// TwinCAT 3 PLC project PLC
// ProgramVersion: 3.1.4026.20
// CompilerDefines: VISU_USEPROPERTYINFO
// libraries:
//   SPT Base Types, * (Beckhoff Automation LLC)
//   SPT Components, * (Beckhoff Automation LLC)
//   SPT Diagnostic, * (Beckhoff Automation LLC)
//   SPT EtherCat, * (Beckhoff Automation LLC)
//   SPT Event Logger, * (Beckhoff Automation LLC)
//   SPT Motion Control, * (Beckhoff Automation LLC)
//   SPT Utilities, * (Beckhoff Automation LLC)
//   Tc2_MC2, * (Beckhoff Automation GmbH)
//   Tc2_MC2_Camming, * (Beckhoff Automation GmbH)
//   Tc2_Standard, * (Beckhoff Automation GmbH)
//   Tc2_System, * (Beckhoff Automation GmbH)
//   Tc2_Utilities, * (Beckhoff Automation GmbH)
//   Tc3_EventLogger, * (Beckhoff Automation GmbH)
//   Tc3_MC2_AdvancedHoming, * (Beckhoff Automation GmbH)
//   Tc3_McCollisionAvoidance, * (Beckhoff Automation GmbH)
//   Tc3_McCoordinatedMotion, * (Beckhoff Automation GmbH)
//   Tc3_PackML_V3, * (Beckhoff Automation GmbH)
// project tree:
//   / GlobalTextList.TcGTLO (not stored), PlcTask.TcTTO (not stored), VisualizationManager.TcVMO (not stored)
//   GVLs/ GVL.TcGVL (not stored)
//   POUs/ Machine.TcPOU, MAIN.TcPOU (not stored)
//   POUs/RackAndPinion/ FB_RackAndPinion.TcPOU
//   VISUs/ Visualization.TcVIS (not stored)
// real-time tasks:
//   TASK PlcTask: cycle T#1ms, priority 20, ADS port 350
//   TASK Job Task: cycle default, priority 32
// motion (NC):
//   TASK NC-Task 1 SAF: cycle T#2ms, priority 4, ADS port 501
//   TASK NC-Task 1 SVB: cycle T#10ms, priority 8, ADS port 511
//   AXIS RnP_Left (id 1)
//     Dynamic: Acceleration=11599.5, Deceleration=11599.5, Jerk=34798.6
//     Velo: RefSearch=10, RefSync=10, SlowManual=1, FastManual=10, Fast=7733.014, Maximum=7733.01
//     OtherSettings: AllowMotionCmdToSlave=true
//     encoder EncType=19
//       EncPara: ScaleFactorNumerator=169.6464, ScaleFactorDenominator=1048576, MaxCount=#xffffffff
//         Inc: RefSearchInverse=true, RefSyncInverse=false, RefPosition=20, RefMode=1
//     drive DrvType=16
//       DrvPara: MaxCount=#xffffffff, DriveControlDWord=#x00020100
//         Analog: VeloReferenz=8506.3154, VeloScale=71.5255737304688, TorqueSetpointScale=10, ScaleFactorActTorque=0.1
//         TimeComp: TaskDelayCycles=1
//     controller CtrType=1
//       CtrPara: PriorControlFactor=1
//         PosDiffControl: Range=15
//         Observer: BandWidth=20
//   AXIS RnP_Right (id 2)
//     Dynamic: Acceleration=11599.521, Deceleration=11599.521, Jerk=34798.563
//     Velo: RefSearch=10, RefSync=10, SlowManual=1, FastManual=10, Fast=7733.014, Maximum=7733.014
//     OtherSettings: AllowMotionCmdToSlave=true
//     encoder EncType=19
//       EncPara: ScaleFactorNumerator=169.6464, ScaleFactorDenominator=1048576, MaxCount=#xffffffff
//         Inc: RefPosition=490, RefMode=6
//     drive DrvType=16
//       DrvPara: MaxCount=#xffffffff, DriveControlDWord=#x00020100
//         Analog: VeloReferenz=8506.3154, VeloScale=71.5255737304688, TorqueSetpointScale=10, ScaleFactorActTorque=0.1
//         TimeComp: TaskDelayCycles=1
//     controller CtrType=1
//       CtrPara: PriorControlFactor=1
//         PosDiffControl: Range=15
//         Observer: BandWidth=20
//   AXIS Ballscrew (id 3)
//     OtherSettings: AllowMotionCmdToSlave=true
//     encoder EncType=19
//       EncPara: MaxCount=#xffffffff
//     drive DrvType=16
//       DrvPara: MaxCount=#xffffffff, DriveControlDWord=#x00000100
//         Analog: TorqueSetpointScale=10, ScaleFactorActTorque=0.1
//         TimeComp: TaskDelayCycles=1
//     controller CtrType=1
//       CtrPara: PriorControlFactor=1
//         Observer: BandWidth=20
// I/O:
//   DEVICE Device 1 (EtherCAT), AmsNetId 169.254.243.188.2.1
//     Term 1 (EK1101) [EK1101 EtherCAT Coupler (2A E-Bus, ID switch)]
//       Term 2 (EL1904) [EL1904, 4 Ch. Safety Input 24V, TwinSAFE]
//         modules: Module 1 (FSOES)
//       Term 3 (EK1110) [EK1110 EtherCAT extension]
//     Term 4 (AX8620-0000-0105) [AX8620-0000-0105]
//       Drive 5 (AX8206-0210-0107) [AX8206-0210-0107 (2Ch. 6A servo axis, safe-motion, multi-FB)]
//         modules: Device, Device, Device, Device, Device, Device, Device, Device, Device, Device, Device (Safety), Device, Device, Device, Device, Device, Device, Device, Device, Device, Device, Device, Device, Device, Device, Device, Device, Device, Device, Device, Device, Ch A, Ch A, Ch A, Ch A, Ch A, Ch A, Ch A, Ch A, Ch A, Ch A, Ch A, Ch A, Ch A, Ch A, Ch A, Ch A, Ch A, Ch A, Ch A, Ch A, Ch A, Ch A, Ch A, Ch A, Ch A, Ch A, Ch B, Ch B, Ch B, Ch B, Ch B, Ch B, Ch B, Ch B, Ch B, Ch B, Ch B, Ch B, Ch B, Ch B, Ch B, Ch B, Ch B, Ch B, Ch B, Ch B, Ch B, Ch B, Ch B, Ch B, Ch B
//         startup 12992:1 := 414D383132312D78467830 // Ch A SynchronousMotor parameters / Configured motor type
//         startup 24768:0 := FEFF // Ch A Interpolation sub mode select
//         startup 13000:5 := 0200 // Ch A SynchronousMotor thermal model / Reaction
//         startup 13000:6 := 0000C841 // Ch A SynchronousMotor thermal model / Partial fraction factor
//         startup 12992:12 := 00803B45 // Ch A SynchronousMotor parameters / Motor rated speed
//         startup 12992:13 := 0000003F // Ch A SynchronousMotor parameters / Motor rated torque
//         startup 24694:0 := F4010000 // Ch A Motor standstill torque
//         startup 24800:0 := D007 // Ch A Positive torque/force limit value
//         startup 24801:0 := D007 // Ch A Negative torque/force limit value
//         startup 12288:6 := 4158383230362D303231302D30303030 // Ch A AxisMain parameters / Configured drive type
//         startup 12867:1 := 00008040 // Ch A TorqueControl parameters / Configured channel rated current
//         startup 12867:2 := 00004041 // Ch A TorqueControl parameters / Configured channel peak current
//         startup 12867:7 := 77BE1F40 // Ch A TorqueControl parameters / Iuvw max sum
//         startup 24672:0 := 08 // Ch A Modes of operation
//         startup 13023:0 := 0000 // Ch A SynchronousMotor control mode
//         startup 12998:1 := CDCCCC3C // Ch A SynchronousMotor commutation monitoring parameters / Speed threshold
//         startup 12864:1 := CAAD2041 // Ch A TorqueControl parameters mappable / Torque control proportional gain q
//         startup 12864:2 := 8A0E7C39 // Ch A TorqueControl parameters mappable / Torque control integral action time q
//         startup 12608:1 := FBD1CD3B // Ch A VelocityControl parameters mappable / Velocity control proportional gain
//         startup 12608:2 := 6F12033C // Ch A VelocityControl parameters mappable / Velocity control integral action time
//         startup 12608:3 := 00980546 // Ch A VelocityControl parameters mappable / Bipolar velocity limit value
//         startup 12992:15 := 0100 // Ch A SynchronousMotor parameters / Motor temperature sensor connection
//         startup 12611:4 := 0400 // Ch A VelocityControl observer / Observer type
//         startup 24672:0 := 08 // Ch A Modes of operation
//         startup 12296:2 := 00 // Ch A AxisMain parameters encoder direction / Primary encoder direction
//       Drive 6 (AX8206-0200-0106) [AX8206-0200-0106 (2Ch. 6A servo axis, safe-motion)]
//         modules: Device, Device, Device, Device, Device, Device, Device, Device, Device, Device, Device (Safety), Device, Device, Device, Device, Device, Device, Device, Device, Device, Device, Device, Device, Device, Device, Device, Device, Device, Device, Device, Device, Ch A, Ch A, Ch A, Ch A, Ch A, Ch A, Ch A, Ch A, Ch A, Ch A, Ch A, Ch A, Ch A, Ch A, Ch A, Ch A, Ch A, Ch A, Ch A, Ch A, Ch A, Ch A, Ch A, Ch A, Ch A, Ch A, Ch A, Ch B, Ch B, Ch B, Ch B, Ch B, Ch B, Ch B, Ch B, Ch B, Ch B, Ch B, Ch B, Ch B, Ch B, Ch B, Ch B, Ch B, Ch B, Ch B, Ch B, Ch B, Ch B, Ch B, Ch B, Ch B, Ch B, Ch B
//         startup 12992:1 := 414D383032322D78447831 // Ch A Motor parameters / Configured motor type
//         startup 24768:0 := FEFF // Ch A Interpolation sub mode select
//         startup 13000:5 := 0200 // Ch A Motor thermal model / Reaction
//         startup 13000:6 := 0000C841 // Ch A Motor thermal model / Partial fraction factor
//         startup 12992:12 := 0000FA45 // Ch A Motor parameters / Motor rated speed
//         startup 12992:13 := E561313F // Ch A Motor parameters / Motor rated torque
//         startup 24694:0 := 20030000 // Ch A Motor standstill torque
//         startup 24800:0 := D007 // Ch A Positive torque/force limit value
//         startup 24801:0 := D007 // Ch A Negative torque/force limit value
//         startup 12288:6 := 4158383230362D303230302D30303030 // Ch A AxisMain parameters / Configured drive type
//         startup 12867:1 := 0000C03F // Ch A TorqueCtrl parameters / Configured channel rated current
//         startup 12867:2 := 00009040 // Ch A TorqueCtrl parameters / Configured channel peak current
//         startup 12867:7 := 77BE1F40 // Ch A TorqueCtrl parameters / Iuvw max sum
//         startup 24672:0 := 08 // Ch A Modes of operation
//         startup 13023:0 := 0000 // Ch A Motor control mode
//         startup 12998:2 := 5D481A3D // Ch A Motor commutation monitoring parameters / Voltage threshold
//         startup 12998:1 := D5B01E3C // Ch A Motor commutation monitoring parameters / Speed threshold
//         startup 12864:1 := 88E9D742 // Ch A TorqueCtrl parameters mappable / Torque control proportional gain q
//         startup 12864:2 := 8A0E7C39 // Ch A TorqueCtrl parameters mappable / Torque control integral action time q
//         startup 12608:1 := 7298793C // Ch A VeloCtrl parameters mappable / Velocity control proportional gain
//         startup 12608:2 := 6F12033C // Ch A VeloCtrl parameters mappable / Velocity control integral action time
//         startup 12608:3 := 00980546 // Ch A VeloCtrl parameters mappable / Bipolar velocity limit value
//         startup 12992:15 := 0100 // Ch A Motor parameters / Motor temperature sensor connection
//         startup 12611:4 := 0400 // Ch A VeloCtrl observer / Observer type
//         startup 24672:0 := 08 // Ch A Modes of operation
//         startup 12296:2 := 00 // Ch A AxisMain parameters encoder direction / Primary encoder direction
//         startup 14016:1 := 414D383032322D78447831 // Ch B Motor parameters / Configured motor type
//         startup 26816:0 := FEFF // Ch B Interpolation sub mode select
//         startup 14024:5 := 0200 // Ch B Motor thermal model / Reaction
//         startup 14024:6 := 0000C841 // Ch B Motor thermal model / Partial fraction factor
//         startup 14016:12 := 0000FA45 // Ch B Motor parameters / Motor rated speed
//         startup 14016:13 := E561313F // Ch B Motor parameters / Motor rated torque
//         startup 26742:0 := 20030000 // Ch B Motor standstill torque
//         startup 26848:0 := D007 // Ch B Positive torque/force limit value
//         startup 26849:0 := D007 // Ch B Negative torque/force limit value
//         startup 13312:6 := 4158383230362D303230302D30303030 // Ch B AxisMain parameters / Configured drive type
//         startup 13891:1 := 0000C03F // Ch B TorqueCtrl parameters / Configured channel rated current
//         startup 13891:2 := 00009040 // Ch B TorqueCtrl parameters / Configured channel peak current
//         startup 13891:7 := 77BE1F40 // Ch B TorqueCtrl parameters / Iuvw max sum
//         startup 26720:0 := 08 // Ch B Modes of operation
//         startup 14047:0 := 0000 // Ch B Motor control mode
//         startup 14022:2 := 5D481A3D // Ch B Motor commutation monitoring parameters / Voltage threshold
//         startup 14022:1 := D5B01E3C // Ch B Motor commutation monitoring parameters / Speed threshold
//         startup 13888:1 := 88E9D742 // Ch B TorqueCtrl parameters mappable / Torque control proportional gain q
//         startup 13888:2 := 8A0E7C39 // Ch B TorqueCtrl parameters mappable / Torque control integral action time q
//         startup 13632:1 := 7298793C // Ch B VeloCtrl parameters mappable / Velocity control proportional gain
//         startup 13632:2 := 6F12033C // Ch B VeloCtrl parameters mappable / Velocity control integral action time
//         startup 13632:3 := 00980546 // Ch B VeloCtrl parameters mappable / Bipolar velocity limit value
//         startup 14016:15 := 0100 // Ch B Motor parameters / Motor temperature sensor connection
//         startup 13635:4 := 0400 // Ch B VeloCtrl observer / Observer type
//         startup 26720:0 := 08 // Ch B Modes of operation
//         startup 13320:2 := 00 // Ch B AxisMain parameters encoder direction / Primary encoder direction
// variable links:
//   NC-Task 1 SAF/Axes/RnP_Left <-> Device 1 (EtherCAT)/Term 4 (AX8620-0000-0105)/Drive 6 (AX8206-0200-0106)
//     Drive/Inputs/In/nDataIn1 <-> Ch A/Ch A PositionControl Inputs/Ch A Following error actual value
//     Drive/Inputs/In/nDataIn3[0] <-> Ch A/Ch A TorqueControl Inputs/Ch A Torque/force actual value
//     Drive/Inputs/In/nDcOutputTime <-> InfoData/DcOutputShift
//     Drive/Inputs/In/nState1 <-> Ch A/Ch A AxisMain Inputs/Ch A Statusword
//     Drive/Inputs/In/nState2 <-> Ch A/Ch A AxisMain Inputs/Ch A Statusword @bit 8
//     Drive/Inputs/In/nState4 @bit 1 <-> WcState/InputToggle0
//     Drive/Inputs/In/nState4 <-> WcState/WcState0
//     Drive/Outputs/Out/nCtrl1 <-> Ch A/Ch A AxisMain Outputs/Ch A Controlword
//     Drive/Outputs/Out/nCtrl2 <-> Ch A/Ch A AxisMain Outputs/Ch A Controlword @bit 8
//     Drive/Outputs/Out/nDataOut1 <-> Ch A/Ch A Interpolator Outputs/Ch A Target position
//     Drive/Outputs/Out/nDataOut2 <-> Ch A/Ch A Interpolator Outputs/Ch A Target velocity
//     Enc/Inputs/In/nDataIn1 <-> Ch A/Ch A AxisMain Inputs/Ch A Position actual value
//     Enc/Inputs/In/nDcInputTime <-> InfoData/DcInputShift
//     Enc/Inputs/In/nState2 @bit 5 <-> Ch A/Ch A AxisMain Inputs/Position actual value invalid
//     Enc/Inputs/In/nState4 @bit 1 <-> WcState/InputToggle0
//     Enc/Inputs/In/nState4 <-> WcState/WcState0
//   NC-Task 1 SAF/Axes/RnP_Right <-> Device 1 (EtherCAT)/Term 4 (AX8620-0000-0105)/Drive 6 (AX8206-0200-0106)
//     Drive/Inputs/In/nDataIn1 <-> Ch B/Ch B PositionControl Inputs/Ch B Following error actual value
//     Drive/Inputs/In/nDataIn3[0] <-> Ch B/Ch B TorqueControl Inputs/Ch B Torque/force actual value
//     Drive/Inputs/In/nDcOutputTime <-> InfoData/DcOutputShift
//     Drive/Inputs/In/nState1 <-> Ch B/Ch B AxisMain Inputs/Ch B Statusword
//     Drive/Inputs/In/nState2 <-> Ch B/Ch B AxisMain Inputs/Ch B Statusword @bit 8
//     Drive/Inputs/In/nState4 @bit 1 <-> WcState/InputToggle0
//     Drive/Inputs/In/nState4 <-> WcState/WcState0
//     Drive/Outputs/Out/nCtrl1 <-> Ch B/Ch B AxisMain Outputs/Ch B Controlword
//     Drive/Outputs/Out/nCtrl2 <-> Ch B/Ch B AxisMain Outputs/Ch B Controlword @bit 8
//     Drive/Outputs/Out/nDataOut1 <-> Ch B/Ch B Interpolator Outputs/Ch B Target position
//     Drive/Outputs/Out/nDataOut2 <-> Ch B/Ch B Interpolator Outputs/Ch B Target velocity
//     Enc/Inputs/In/nDataIn1 <-> Ch B/Ch B AxisMain Inputs/Ch B Position actual value
//     Enc/Inputs/In/nDcInputTime <-> InfoData/DcInputShift
//     Enc/Inputs/In/nState2 @bit 5 <-> Ch B/Ch B AxisMain Inputs/Position actual value invalid
//     Enc/Inputs/In/nState4 @bit 1 <-> WcState/InputToggle0
//     Enc/Inputs/In/nState4 <-> WcState/WcState0
//   PLC/PLC Instance <-> Device 1 (EtherCAT)/Term 4 (AX8620-0000-0105)/Drive 5 (AX8206-0210-0107)
//     PlcTask Inputs/MAIN.SafetyEstop.InfoData/Diag <-> Device (Safety)/Function Block Info Data/TwinSafeGroup1.Network1.FBEstop1 Info Data/Diag
//     PlcTask Inputs/MAIN.SafetyEstop.InfoData/State <-> Device (Safety)/Function Block Info Data/TwinSafeGroup1.Network1.FBEstop1 Info Data/State
//     PlcTask Inputs/MAIN.SafetyGroup_Main.InfoData/Diag <-> Device (Safety)/Group Info Data/TwinSafeGroup1 Info Data/Diag
//     PlcTask Inputs/MAIN.SafetyGroup_Main.InfoData/State <-> Device (Safety)/Group Info Data/TwinSafeGroup1 Info Data/State
//     PlcTask Inputs/MAIN.SafetyOK <-> Device (Safety)/Standard Inputdata/Standard Out Var 7
//     PlcTask Outputs/MAIN.SafetyFBReset <-> Device (Safety)/Standard Outputdata/Standard In Var 6
//     PlcTask Outputs/MAIN.SafetyGroupAutoReset.Reset <-> Device (Safety)/Standard Outputdata/Standard In Var 1
//     PlcTask Outputs/MAIN.SafetyGroup_Main.Run <-> Device (Safety)/Standard Outputdata/Standard In Var 2
//   PLC/PLC Instance <-> NC-Task 1 SAF/Axes/RnP_Left
//     PlcTask Inputs/MAIN.Machine.RackAndPinion.LeftAxis.BasicAxis._Axis.NcToPlc <-> Outputs/ToPlc
//     PlcTask Outputs/MAIN.Machine.RackAndPinion.LeftAxis.BasicAxis._Axis.PlcToNc <-> Inputs/FromPlc
//   PLC/PLC Instance <-> NC-Task 1 SAF/Axes/RnP_Right
//     PlcTask Inputs/MAIN.Machine.RackAndPinion.RightAxis.BasicAxis._Axis.NcToPlc <-> Outputs/ToPlc
//     PlcTask Outputs/MAIN.Machine.RackAndPinion.RightAxis.BasicAxis._Axis.PlcToNc <-> Inputs/FromPlc
//   PLC/PLC Instance <-> NC-Task 1 SAF/Objects/Group1 (CA Group)
//     PlcTask Inputs/MAIN.Machine.RackAndPinion.CAGroup.NcToPlc <-> Group Outputs/ToPLC
//     PlcTask Outputs/MAIN.Machine.RackAndPinion.CAGroup.PlcToNc/CA <-> Group Inputs/FromPLC
//   (this object) <-> Device 1 (EtherCAT)/Term 4 (AX8620-0000-0105)/Drive 5 (AX8206-0210-0107)
//     Drive/Inputs/In/nDataIn1 <-> Ch A/Ch A PositionControl Inputs/Ch A Following error actual value
//     Drive/Inputs/In/nDataIn3[0] <-> Ch A/Ch A TorqueControl Inputs/Ch A Torque/force actual value
//     Drive/Inputs/In/nDcOutputTime <-> InfoData/DcOutputShift
//     Drive/Inputs/In/nState1 <-> Ch A/Ch A AxisMain Inputs/Ch A Statusword
//     Drive/Inputs/In/nState2 <-> Ch A/Ch A AxisMain Inputs/Ch A Statusword @bit 8
//     Drive/Inputs/In/nState4 @bit 1 <-> WcState/InputToggle0
//     Drive/Inputs/In/nState4 <-> WcState/WcState0
//     Drive/Outputs/Out/nCtrl1 <-> Ch A/Ch A AxisMain Outputs/Ch A Controlword
//     Drive/Outputs/Out/nCtrl2 <-> Ch A/Ch A AxisMain Outputs/Ch A Controlword @bit 8
//     Drive/Outputs/Out/nDataOut1 <-> Ch A/Ch A Interpolator Outputs/Ch A Target position
//     Drive/Outputs/Out/nDataOut2 <-> Ch A/Ch A Interpolator Outputs/Ch A Target velocity
//     Enc/Inputs/In/nDataIn1 <-> Ch A/Ch A AxisMain Inputs/Ch A Position actual value
//     Enc/Inputs/In/nDcInputTime <-> InfoData/DcInputShift
//     Enc/Inputs/In/nState2 @bit 5 <-> Ch A/Ch A AxisMain Inputs/Position actual value invalid
//     Enc/Inputs/In/nState4 @bit 1 <-> WcState/InputToggle0
//     Enc/Inputs/In/nState4 <-> WcState/WcState0
//   (this object) <-> Device 1 (EtherCAT)
//     Term 1 (EK1101)/Term 2 (EL1904)/Module 1 (FSOES)/RxPDO/FSOE <-> Term 4 (AX8620-0000-0105)/Drive 5 (AX8206-0210-0107)/Device (Safety)/FSoE Master Connection 1 Master Message/Message_3
//     Term 1 (EK1101)/Term 2 (EL1904)/Module 1 (FSOES)/TxPDO/FSOE <-> Term 4 (AX8620-0000-0105)/Drive 5 (AX8206-0210-0107)/Device (Safety)/FSoE Master Connection 1 Slave Message/Message_3
//     Term 4 (AX8620-0000-0105)/Drive 5 (AX8206-0210-0107)/Device (Safety)/FSoE Master Connection 1 Master Message/Message_3 <-> Term 1 (EK1101)/Term 2 (EL1904)/Module 1 (FSOES)/RxPDO/FSOE
//     Term 4 (AX8620-0000-0105)/Drive 5 (AX8206-0210-0107)/Device (Safety)/FSoE Master Connection 1 Slave Message/Message_3 <-> Term 1 (EK1101)/Term 2 (EL1904)/Module 1 (FSOES)/TxPDO/FSOE
//     Term 4 (AX8620-0000-0105)/Drive 5 (AX8206-0210-0107)/Device (Safety)/FSoE Master Connection 2 Master Message/Message_5 <-> Term 4 (AX8620-0000-0105)/Drive 6 (AX8206-0200-0106)/Device (Safety)/FSoE Slave Connection 1 Master Message/FSOE
//     Term 4 (AX8620-0000-0105)/Drive 5 (AX8206-0210-0107)/Device (Safety)/FSoE Master Connection 2 Slave Message/Message_5 <-> Term 4 (AX8620-0000-0105)/Drive 6 (AX8206-0200-0106)/Device (Safety)/FSoE Slave Connection 1 Slave Message/FSOE
//     Term 4 (AX8620-0000-0105)/Drive 5 (AX8206-0210-0107)/Device/DeviceMain Outputs/Power supply controlword <-> Term 4 (AX8620-0000-0105)/PSM Controlword for axis/Controlword for axis
//     Term 4 (AX8620-0000-0105)/Drive 6 (AX8206-0200-0106)/Device/DeviceMain Outputs/Power supply controlword <-> Term 4 (AX8620-0000-0105)/PSM Controlword for axis/Controlword for axis
//     Term 4 (AX8620-0000-0105)/Drive 6 (AX8206-0200-0106)/Device (Safety)/FSoE Slave Connection 1 Master Message/FSOE <-> Term 4 (AX8620-0000-0105)/Drive 5 (AX8206-0210-0107)/Device (Safety)/FSoE Master Connection 2 Master Message/Message_5
//     Term 4 (AX8620-0000-0105)/Drive 6 (AX8206-0200-0106)/Device (Safety)/FSoE Slave Connection 1 Slave Message/FSOE <-> Term 4 (AX8620-0000-0105)/Drive 5 (AX8206-0210-0107)/Device (Safety)/FSoE Master Connection 2 Slave Message/Message_5
//     Term 4 (AX8620-0000-0105)/PSM Controlword for axis/Controlword for axis <-> Term 4 (AX8620-0000-0105)/Drive 5 (AX8206-0210-0107)/Device/DeviceMain Outputs/Power supply controlword
//     Term 4 (AX8620-0000-0105)/PSM Controlword for axis/Controlword for axis <-> Term 4 (AX8620-0000-0105)/Drive 6 (AX8206-0200-0106)/Device/DeviceMain Outputs/Power supply controlword

// ---- POUs/Machine.TcPOU
FUNCTION_BLOCK Machine EXTENDS FB_PackML_BaseModule
VAR
	RackAndPinion	: FB_RackAndPinion;
END_VAR

METHOD PROTECTED HMIPermissions
AllowHMIControl(TRUE);
END_METHOD

(* Basic module initialization logic*)
METHOD PROTECTED Initialize : BOOL
Initialize := FALSE;
CASE DescendantSequenceState OF
	0:
		RegisterSubmodule(SubModule := RackAndPinion);
		DescendantSequenceState := DescendantSequenceState + 10;

	10:
		IF SUPER^.Initialize() THEN
			Initialize := TRUE;
		END_IF
END_CASE
END_METHOD

END_FUNCTION_BLOCK

// ---- POUs/RackAndPinion/FB_RackAndPinion.TcPOU
FUNCTION_BLOCK FB_RackAndPinion EXTENDS FB_PackML_BaseModule
VAR
	LeftAxis	: FB_Component_BasicAxis;
	RightAxis	: FB_Component_BasicAxis;

	// CA Group
	CAGroup			: AXES_GROUP_REF;
	GroupReadStatus	: MC_GroupReadStatus;
	GroupReset		: MC_GroupReset;
	GroupEnable		: MC_GroupEnable;
	GroupDisable	: MC_GroupDisable;
	AddToGroup		: ARRAY[0..1] OF MC_AddAxisToGroup;
	MoveAbsoluteCA	: ARRAY[0..1] OF MC_MoveAbsoluteCA;

	TON_Dwell	: TON;
END_VAR

//! @summary This method contains code which will execute when this PackML module is in the <b>Aborting</b> state
METHOD PROTECTED Aborting
VAR
	i				: UDINT;
	SubModulesReady : BOOL := TRUE;
END_VAR
CASE DescendantSequenceState OF
	0:
		NoStateTasksToComplete := FALSE;
		DescendantSequenceState := DescendantSequenceState + 10;

	10:
		IF LeftAxis.Disable() AND RightAxis.Disable() THEN
			StateTasksComplete 		:= TRUE;
			DescendantSequenceState := DescendantSequenceState + 10;
		END_IF

	//20:	

	20:
		StateTasksComplete := TRUE;
END_CASE

SUPER^.Aborting();
END_METHOD

//! @summary This method contains code which will execute when this PackML module is in the <b>Clearing</b> state
METHOD PROTECTED Clearing
VAR
	i				: UDINT;
	SubModulesReady : BOOL := TRUE;
END_VAR

VAR_INST

END_VAR

(*! <description> <b>Note:</b> The <i>Clear</i> command can also be thought of as a <i>fault reset</i> depite the ambiguity in the naming of the <i>Reset</i> state. 
<table> 
	<tr>
		<th> Previous State </th>
		<th> Transition In </th>
		<th> Transition Out </th>
		<th> Next State  </th> 
	</tr>
	<tr>
		<td> Aborted </td>
		<td> Clear Command </td> 
		<td> State Complete </td>
		<td> Stopped </td> 
	</tr>
</table>
This method is called as required by <c>StateControl()</c>
</description> 

*)
// CASE _CurrentMode OF
// 	E_PMLUnitMode.ePMLUnitMode_Production:
		CASE DescendantSequenceState OF
			0: //Init
				NoStateTasksToComplete := FALSE;

				//Reset Axes and  CA Group
				LeftAxis.Reset();
				RightAxis.Reset();
				GroupReset.Execute	:= TRUE;
				DescendantSequenceState := DescendantSequenceState + 10;

			10: // Done	
				GroupReset.Execute	:= FALSE;
				StateTasksComplete := TRUE;
		END_CASE

// END_CASE

SUPER^.Clearing();
END_METHOD

METHOD CyclicLogic
VAR_INPUT
END_VAR
SUPER^.CyclicLogic();

AddToGroup[0](Axis := LeftAxis.Axis, AxesGroup := CAGroup);
AddToGroup[1](Axis := RightAxis.Axis, AxesGroup := CAGroup);
GroupEnable(AxesGroup := CAGroup);
GroupDisable(AxesGroup := CAGroup);
GroupReadStatus.Enable		:= TRUE;
GroupReadStatus(AxesGroup	:= CAGroup);
GroupReset(AxesGroup	:= CAGroup);
MoveAbsoluteCA[0](Axis := LeftAxis.Axis);
MoveAbsoluteCA[1](Axis := RightAxis.Axis);
TON_Dwell();
END_METHOD

//! @summary This method contains code which will execute when this PackML module is in the <b>Execute</b> state
METHOD PROTECTED Execute
VAR
	i : UDINT;
END_VAR
(*CASE _CurrentMode OF
	E_PMLUnitMode.ePMLUnitMode_Production:


	E_PMLUnitMode.ePMLUnitMode_Manual:
		; //Insert logic for Manual Mode here
END_CASE	*)

CASE DescendantSequenceState OF
	0:
		FOR i := 0 TO 1 DO
			MoveAbsoluteCA[i].Execute		:= TRUE;
			MoveAbsoluteCA[i].Position		:= 50.0;
			MoveAbsoluteCA[i].Velocity		:= leftAxis.Velocity;
			MoveAbsoluteCA[i].Acceleration	:= LeftAxis.Acceleration;
			MoveAbsoluteCA[i].Deceleration	:= LeftAxis.Deceleration;
			MoveAbsoluteCA[i].Jerk			:= LeftAxis.Jerk;
			MoveAbsoluteCA[i].Gap			:= 68.0;
			MoveAbsoluteCA[i].Options.GapControlMode	:= MC_GAP_CONTROL_MODE.mcGapControlModeFast;
			MoveAbsoluteCA[i].BufferMode	:= mcAborting;
		END_FOR
		DescendantSequenceState				:= DescendantSequenceState + 10;

	10:	IF MoveAbsoluteCA[0].Done OR MoveAbsoluteCA[1].Done THEN
			MoveAbsoluteCA[0].Execute		:= FALSE;
			MoveAbsoluteCA[1].Execute		:= FALSE;
			TON_Dwell.IN	:= TRUE;
			TON_Dwell.PT	:= T#1S;
			DescendantSequenceState			:= DescendantSequenceState + 10;
		END_IF

	20: IF TON_Dwell.Q THEN
			ton_dwell.IN	:= FALSE;
			DescendantSequenceState			:= DescendantSequenceState + 10;
		END_IF

	30:
		FOR i := 0 TO 1 DO
			MoveAbsoluteCA[i].Execute		:= TRUE;
			MoveAbsoluteCA[i].Position		:= 450.0;
			MoveAbsoluteCA[i].Velocity		:= leftAxis.Velocity;
			MoveAbsoluteCA[i].Acceleration	:= LeftAxis.Acceleration;
			MoveAbsoluteCA[i].Deceleration	:= LeftAxis.Deceleration;
			MoveAbsoluteCA[i].Jerk			:= LeftAxis.Jerk;
			MoveAbsoluteCA[i].Gap			:= 68.0;
			MoveAbsoluteCA[i].Options.GapControlMode	:= MC_GAP_CONTROL_MODE.mcGapControlModeStandard;
			MoveAbsoluteCA[i].BufferMode	:= mcAborting;
		END_FOR
		DescendantSequenceState				:= DescendantSequenceState + 10;

	40:	IF MoveAbsoluteCA[0].Done OR MoveAbsoluteCA[1].Done THEN
			MoveAbsoluteCA[0].Execute		:= FALSE;
			MoveAbsoluteCA[1].Execute		:= FALSE;
			TON_Dwell.IN	:= TRUE;
			TON_Dwell.PT	:= T#1S;
			DescendantSequenceState			:= DescendantSequenceState + 10;

		END_IF

	50: IF TON_Dwell.Q THEN
			ton_dwell.IN	:= FALSE;
			DescendantSequenceState			:= 0;
		END_IF

END_CASE
END_METHOD

(* Basic module initialization logic*)
METHOD PROTECTED Initialize : BOOL
Initialize := FALSE;
CASE DescendantSequenceState OF
	0:
		RegisterComponent(Component := LeftAxis);
		RegisterComponent(Component := RightAxis);
		DescendantSequenceState := DescendantSequenceState + 10;

	10:
		IF SUPER^.Initialize() THEN
			DescendantSequenceState := DescendantSequenceState + 10;
		END_IF

	20:
		Initialize := TRUE;
END_CASE
END_METHOD

METHOD PROTECTED Resetting
VAR_INST
	i			 : UDINT;
END_VAR
// CASE _CurrentMode OF
// 	E_PMLUnitMode.ePMLUnitMode_Production:
		CASE DescendantSequenceState OF
			0: //Init
				i					   := 1;
				NoStateTasksToComplete := FALSE;
				DescendantSequenceState := DescendantSequenceState + 10;

			10: //Enable Axes
				IF LeftAxis.Enable() AND RightAxis.Enable() THEN
					DescendantSequenceState := DescendantSequenceState + 10;
				END_IF

			// Add logic to home left axis to switch and right axis to hard stop
			20: // Home Right Axis


			30:	// Home Left Axis


			40: //Add Movers to Group			
				AddToGroup[0].Execute		:= AddToGroup[1].Execute		:= TRUE;
				AddToGroup[0].IdentInGroup	:= UDINT_TO_IDENTINGROUP(1);
				AddToGroup[1].IdentInGroup	:= UDINT_TO_IDENTINGROUP(2);
				IF AddToGroup[0].Done AND AddToGroup[1].Done THEN	
					AddToGroup[0].Execute	:= AddToGroup[1].Execute	:= FALSE;
					DescendantSequenceState := DescendantSequenceState + 10;
				END_IF

			50: //Enable CA Group
				GroupEnable.Execute	:= TRUE;
				IF GroupEnable.Done THEN
					DescendantSequenceState := DescendantSequenceState + 10;
				END_IF

			60: //Clearing complete
				StateTasksComplete := TRUE;

		END_CASE
// END_CASE

SUPER^.Resetting();
END_METHOD

METHOD PROTECTED Starting
VAR_INST
	i		  : UDINT;
END_VAR
//CASE _CurrentMode OF
//	E_PMLUnitMode.ePMLUnitMode_Production:
		CASE DescendantSequenceState OF
			0:
				NoStateTasksToComplete	:= FALSE;
				DescendantSequenceState := 10;
				i						:= 1;

			10: //Set Axis Parameters
				LeftAxis.Velocity		:= 250;		RightAxis.Velocity		:= 250;
				LeftAxis.Acceleration	:= 1000;	RightAxis.Acceleration	:= 1000;
				LeftAxis.Deceleration	:= 1000;	RightAxis.Deceleration	:= 1000;
				LeftAxis.Jerk			:= 10000;	RightAxis.Jerk			:= 10000;
				DescendantSequenceState := DescendantSequenceState + 10;
				StateTasksComplete 		:= TRUE;

			20: //Cleanup mover queues
				DescendantSequenceState := DescendantSequenceState + 10;

		END_CASE

	//E_PMLUnitMode.ePMLUnitMode_Manual:
//END_CASE

SUPER^.Starting();
END_METHOD

END_FUNCTION_BLOCK
